% RSLogix 500 project TRAFFIC LIGHT STOP.RSS, saved by version 8.30.00.16 %
PROJECT "UNTITLED"    % processor: MicroLogix 1000 %

PROGRAM FILES
  LAD 2 "MAIN_PROG"  11 rungs
  LAD 3 "USER_FAULT"  1 rungs
  LAD 4 "HSC_INT"  1 rungs
  LAD 5 "STI_INT"  1 rungs
  LAD 6, 7, 8, 9, 10, 11, 12, 13, 14, 15, 16: only END

DATA FILES
  O0 OUTPUT  1 elements
  I1 INPUT  2 elements
  S2 STATUS  33 elements
  B3 BINARY  32 elements
  T4 TIMER  40 elements
  C5 COUNTER  32 elements
  R6 CONTROL  16 elements
  N7 INTEGER  105 elements

LADDER 2 "MAIN_PROG"
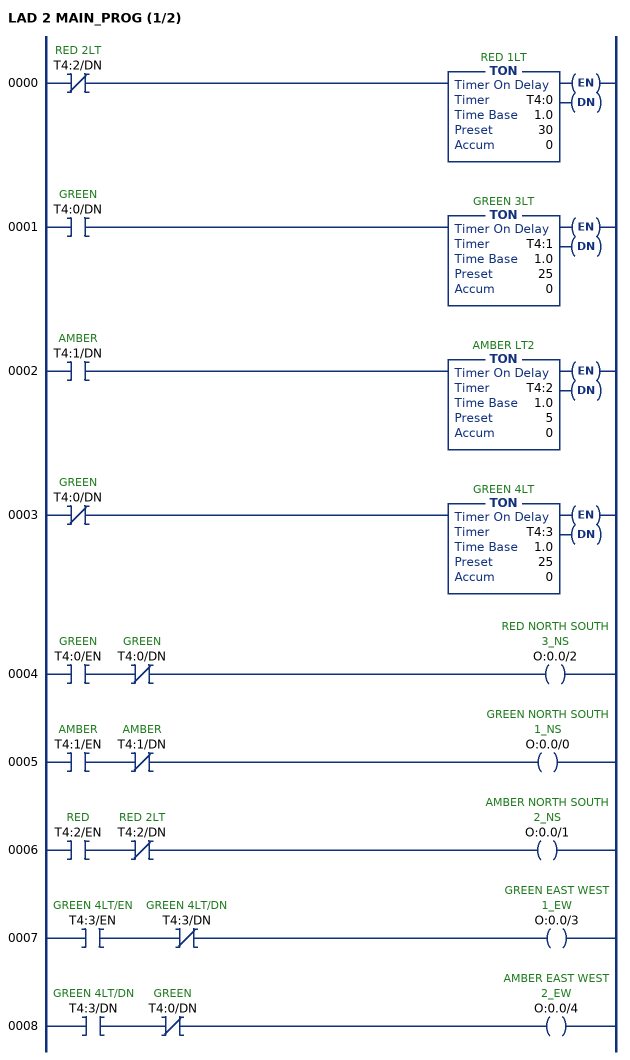
% Rung: 0 %
SOR XIO T4:2/DN TON T4:0 1.0 30 0 EOR
%   T4:2/DN  2LT  "RED" %
%   T4:0  1LT  "RED" %
% Rung: 1 %
SOR XIC T4:0/DN TON T4:1 1.0 25 0 EOR
%   T4:0/DN  "GREEN" %
%   T4:1  3LT  "GREEN" %
% Rung: 2 %
SOR XIC T4:1/DN TON T4:2 1.0 5 0 EOR
%   T4:1/DN  "AMBER" %
%   T4:2  LT2  "AMBER" %
% Rung: 3 %
SOR XIO T4:0/DN TON T4:3 1.0 25 0 EOR
%   T4:0/DN  "GREEN" %
%   T4:3  4LT  "GREEN" %
% Rung: 4 %
SOR XIC T4:0/EN XIO T4:0/DN OTE O:0.0/2 EOR
%   T4:0/EN  "GREEN" %
%   T4:0/DN  "GREEN" %
%   O:0.0/2  3_NS  "RED NORTH SOUTH" %
% Rung: 5 %
SOR XIC T4:1/EN XIO T4:1/DN OTE O:0.0/0 EOR
%   T4:1/EN  "AMBER" %
%   T4:1/DN  "AMBER" %
%   O:0.0/0  1_NS  "GREEN NORTH SOUTH" %
% Rung: 6 %
SOR XIC T4:2/EN XIO T4:2/DN OTE O:0.0/1 EOR
%   T4:2/EN  "RED" %
%   T4:2/DN  2LT  "RED" %
%   O:0.0/1  2_NS  "AMBER NORTH SOUTH" %
% Rung: 7 %
SOR XIC T4:3/EN XIO T4:3/DN OTE O:0.0/3 EOR
%   T4:3  4LT  "GREEN" %
%   O:0.0/3  1_EW  "GREEN EAST WEST" %
% Rung: 8 %
SOR XIC T4:3/DN XIO T4:0/DN OTE O:0.0/4 EOR
%   T4:3  4LT  "GREEN" %
%   T4:0/DN  "GREEN" %
%   O:0.0/4  2_EW  "AMBER EAST WEST" %

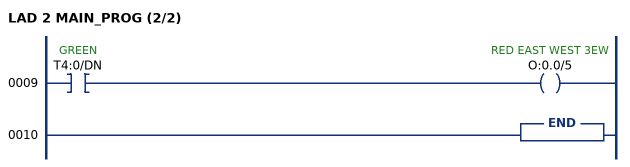
% Rung: 9 %
SOR XIC T4:0/DN OTE O:0.0/5 EOR
%   T4:0/DN  "GREEN" %
%   O:0.0/5  3EW  "RED EAST WEST" %
% Rung: 10 %
SOR END EOR

DATA TABLE (non-zero values as saved)
DATA T4
% .PRE .ACC %
% T4:0 % 30 0
% T4:1 % 25 0
% T4:2 % 5 0
% T4:3 % 25 0
